TYPE strQueueDetail :
	STRUCT
		uiPrio			: UINT;				(* Option Sendepriorität 				*)
		uiMsgHandle 	: UDINT;			(* unique msg handle,  					*)
		pDATA			: POINTER TO BYTE ;	(* pointer on real data 				*)
		szDATA			: UDINT;			(* Length of data from pointer reference*)
	END_STRUCT
END_TYPE

(* stored: Version 1.1.0.1, ProductVersion 3.1.4024.12
   DUT strQueueDetail: Id {4ec66aaa-2b50-42ad-a9f4-c01b840339a1} *)
